// TIA Portal V19 export
FUNCTION "AFC_DelayON" : Void   // FC2, FBD
TITLE = AFC_DELAYON
{ S7_Optimized_Access := 'TRUE' }
AUTHOR : CH
FAMILY : Aktina
NAME : Global
// AFC_DELAYON
// stored: AutoNumber false, IsIECCheckEnabled true, SetENOAutomatically false
   VAR_INPUT
      cmd : Bool;   // Command run
      Pulse : Bool;   // 100ms pulse
      Reset : Bool;   // Reset immediately
   END_VAR
   VAR_OUTPUT
      on : Bool;   // Activation
   END_VAR
   VAR_IN_OUT
      Data : Variant;   // Data area
   END_VAR
   VAR_TEMP
      i : "UDT_DELAYON";   // Local stack
      logical1 : Bool;   // Logical 1
      calc : Real;   // Calculation intermediate
   END_VAR
BEGIN

REGION Network 1: GEN: Set Logical 1
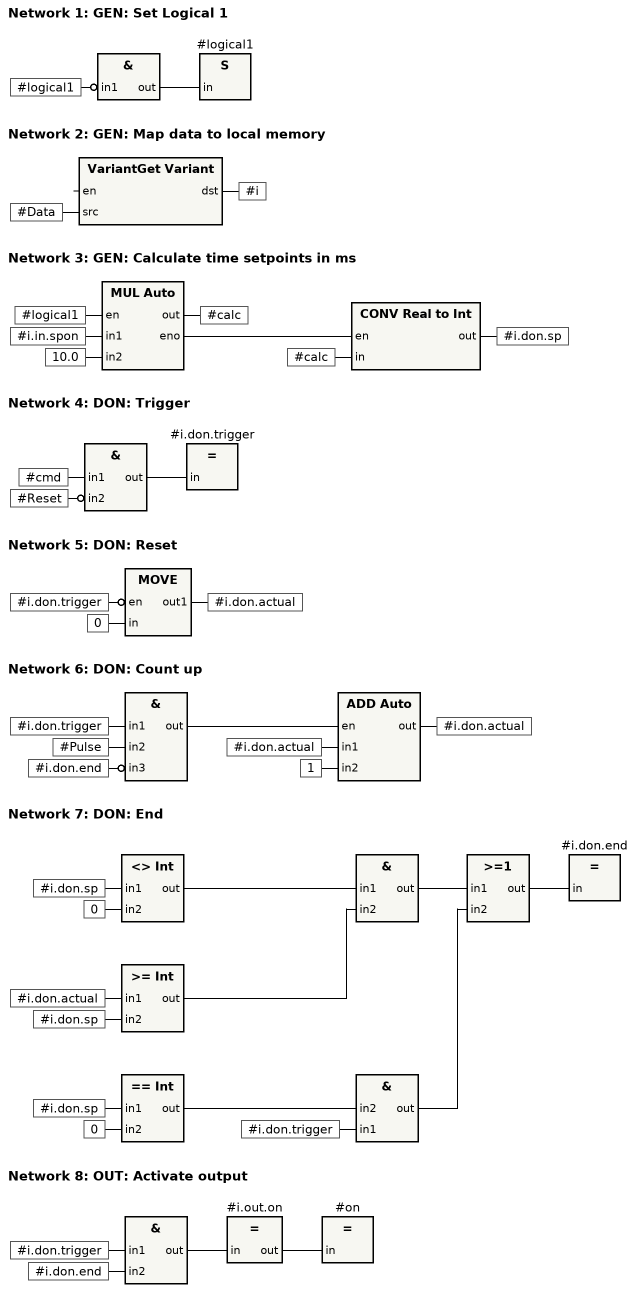
   IF NOT #logical1 THEN #logical1 := TRUE; END_IF;
END_REGION

REGION Network 2: GEN: Map data to local memory
   // no SCL statement known for VariantGet: written as a call
   VariantGet(src := #Data, dst => #i);
END_REGION

REGION Network 3: GEN: Calculate time setpoints in ms
   IF #logical1 THEN
       #calc := #i.in.spon * 10.0;
       #i.don.sp := REAL_TO_INT(#calc);
   END_IF;
END_REGION

REGION Network 4: DON: Trigger
   #i.don.trigger := #cmd AND NOT #Reset;
END_REGION

REGION Network 5: DON: Reset
   IF NOT #i.don.trigger THEN #i.don.actual := 0; END_IF;
END_REGION

REGION Network 6: DON: Count up
   IF #i.don.trigger AND #Pulse AND NOT #i.don.end THEN #i.don.actual := #i.don.actual + 1; END_IF;
END_REGION

REGION Network 7: DON: End
   #i.don.end := ((#i.don.sp <> 0) AND (#i.don.actual >= #i.don.sp)) OR ((#i.don.sp = 0) AND #i.don.trigger);
END_REGION

REGION Network 8: OUT: Activate output
   #i.out.on := #i.don.trigger AND #i.don.end;
   #on := #i.out.on;
END_REGION

REGION Network 9: GEN: Export data to db
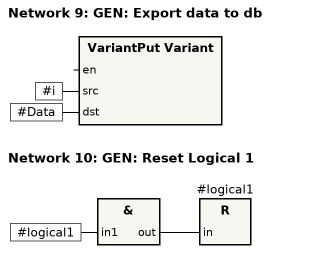
   // no SCL statement known for VariantPut: written as a call
   VariantPut(src := #i, dst := #Data);
END_REGION

REGION Network 10: GEN: Reset Logical 1
   IF #logical1 THEN #logical1 := FALSE; END_IF;
END_REGION
END_FUNCTION
